FUNCTION_BLOCK PUBLIC BYTE_TO_TestSuite EXTENDS TcUnit.FB_TestSuite
VAR
END_VAR

Check_BYTE_TO_BOOL_Max();
Check_BYTE_TO_BOOL_Min();
Check_BYTE_TO_BYTE_Max();
Check_BYTE_TO_BYTE_Min();
Check_BYTE_TO_WORD_Max();
Check_BYTE_TO_WORD_Min();
Check_BYTE_TO_DWORD_Max();
Check_BYTE_TO_DWORD_Min();
Check_BYTE_TO_LWORD_Max();
Check_BYTE_TO_LWORD_Min();
Check_BYTE_TO_SINT_Max();
Check_BYTE_TO_SINT_Min();
Check_BYTE_TO_SINT_TooHigh();
Check_BYTE_TO_INT_Max();
Check_BYTE_TO_INT_Min();
Check_BYTE_TO_DINT_Max();
Check_BYTE_TO_DINT_Min();
Check_BYTE_TO_LINT_Max();
Check_BYTE_TO_LINT_Min();
Check_BYTE_TO_USINT_Max();
Check_BYTE_TO_USINT_Min();
Check_BYTE_TO_UINT_Max();
Check_BYTE_TO_UINT_Min();
Check_BYTE_TO_UDINT_Max();
Check_BYTE_TO_UDINT_Min();
Check_BYTE_TO_ULINT_Max();
Check_BYTE_TO_ULINT_Min();
Check_BYTE_TO_REAL_Max();
Check_BYTE_TO_REAL_Min();
Check_BYTE_TO_LREAL_Max();
Check_BYTE_TO_LREAL_Min();
Check_BYTE_TO_TIME_Max();
Check_BYTE_TO_TIME_Min();
Check_BYTE_TO_TOD_Max();
Check_BYTE_TO_TOD_Min();
Check_BYTE_TO_DATE_Max();
Check_BYTE_TO_DATE_Min();
Check_BYTE_TO_DT_Max();
Check_BYTE_TO_DT_Min();
Check_BYTE_TO_STRING_Max();
Check_BYTE_TO_STRING_Min();

METHOD PUBLIC Check_BYTE_TO_BOOL_Min
VAR
	value : BYTE := DatatypeLimits.BYTE_MIN_VALUE;
	actual : BOOL;
	converted : BOOL;
	equal : BOOL;
END_VAR
TEST('Check_BYTE_TO_BOOL_Min');

// @TEST-RUN
converted := TryConvert_BYTE_TO_Destination(value, actual);
equal := actual = BYTE_TO_BOOL(value);

// @TEST-ASSERT
AssertTrue(Condition := equal, Message := 'Did not convert BYTE to BOOL correctly');
AssertTrue(Condition := converted, Message := 'Did not report BYTE to BOOL conversion was successful');

TEST_FINISHED();
END_METHOD

METHOD PUBLIC Check_BYTE_TO_BOOL_Max
VAR
	value : BYTE := DatatypeLimits.BYTE_MAX_VALUE;
	actual : BOOL;
	converted : BOOL;
	equal : BOOL;
END_VAR
TEST('Check_BYTE_TO_BOOL_Max');

// @TEST-RUN
converted := TryConvert_BYTE_TO_Destination(value, actual);
equal := actual = BYTE_TO_BOOL(value);

// @TEST-ASSERT
AssertTrue(Condition := equal, Message := 'Did not convert BYTE to BOOL correctly');
AssertTrue(Condition := converted, Message := 'Did not report BYTE to BOOL conversion was successful');

TEST_FINISHED();
END_METHOD

METHOD PUBLIC Check_BYTE_TO_BYTE_Min
VAR
	value : BYTE := DatatypeLimits.BYTE_MIN_VALUE;
	actual : BYTE;
	converted : BOOL;
	equal : BOOL;
END_VAR
TEST('Check_BYTE_TO_BYTE_Min');

// @TEST-RUN
converted := TryConvert_BYTE_TO_Destination(value, actual);
equal := actual = value;

// @TEST-ASSERT
AssertTrue(Condition := equal, Message := 'Did not convert BYTE to BYTE correctly');
AssertTrue(Condition := converted, Message := 'Did not report BYTE to BYTE conversion was successful');

TEST_FINISHED();
END_METHOD

METHOD PUBLIC Check_BYTE_TO_BYTE_Max
VAR
	value : BYTE := DatatypeLimits.BYTE_MAX_VALUE;
	actual : BYTE;
	converted : BOOL;
	equal : BOOL;
END_VAR
TEST('Check_BYTE_TO_BYTE_Max');

// @TEST-RUN
converted := TryConvert_BYTE_TO_Destination(value, actual);
equal := actual = value;

// @TEST-ASSERT
AssertTrue(Condition := equal, Message := 'Did not convert BYTE to BYTE correctly');
AssertTrue(Condition := converted, Message := 'Did not report BYTE to BYTE conversion was successful');

TEST_FINISHED();
END_METHOD

METHOD PUBLIC Check_BYTE_TO_DATE_Min
VAR
	value : BYTE := DatatypeLimits.BYTE_MIN_VALUE;
	actual : DATE;
	converted : BOOL;
	equal : BOOL;
END_VAR
TEST('Check_BYTE_TO_DATE_Min');

// @TEST-RUN
converted := TryConvert_BYTE_TO_Destination(value, actual);
equal := actual = BYTE_TO_DATE(value);

// @TEST-ASSERT
AssertTrue(Condition := equal, Message := 'Did not convert BYTE to DATE correctly');
AssertTrue(Condition := converted, Message := 'Did not report BYTE to DATE conversion was successful');

TEST_FINISHED();
END_METHOD

METHOD PUBLIC Check_BYTE_TO_DATE_Max
VAR
	value : BYTE := DatatypeLimits.BYTE_MAX_VALUE;
	actual : DATE;
	converted : BOOL;
	equal : BOOL;
END_VAR
TEST('Check_BYTE_TO_DATE_Max');

// @TEST-RUN
converted := TryConvert_BYTE_TO_Destination(value, actual);
equal := actual = BYTE_TO_DATE(value);

// @TEST-ASSERT
AssertTrue(Condition := equal, Message := 'Did not convert BYTE to DATE correctly');
AssertTrue(Condition := converted, Message := 'Did not report BYTE to DATE conversion was successful');

TEST_FINISHED();
END_METHOD

METHOD PUBLIC Check_BYTE_TO_DINT_Min
VAR
	value : BYTE := DatatypeLimits.BYTE_MIN_VALUE;
	actual : DINT;
	converted : BOOL;
	equal : BOOL;
END_VAR
TEST('Check_BYTE_TO_DINT_Min');

// @TEST-RUN
converted := TryConvert_BYTE_TO_Destination(value, actual);
equal := actual = BYTE_TO_DINT(value);

// @TEST-ASSERT
AssertTrue(Condition := equal, Message := 'Did not convert BYTE to DINT correctly');
AssertTrue(Condition := converted, Message := 'Did not report BYTE to DINT conversion was successful');

TEST_FINISHED();
END_METHOD

METHOD PUBLIC Check_BYTE_TO_DINT_Max
VAR
	value : BYTE := DatatypeLimits.BYTE_MAX_VALUE;
	actual : DINT;
	converted : BOOL;
	equal : BOOL;
END_VAR
TEST('Check_BYTE_TO_DINT_Max');

// @TEST-RUN
converted := TryConvert_BYTE_TO_Destination(value, actual);
equal := actual = BYTE_TO_DINT(value);

// @TEST-ASSERT
AssertTrue(Condition := equal, Message := 'Did not convert BYTE to DINT correctly');
AssertTrue(Condition := converted, Message := 'Did not report BYTE to DINT conversion was successful');

TEST_FINISHED();
END_METHOD

METHOD PUBLIC Check_BYTE_TO_DT_Min
VAR
	value : BYTE := DatatypeLimits.BYTE_MIN_VALUE;
	actual : DT;
	converted : BOOL;
	equal : BOOL;
END_VAR
TEST('Check_BYTE_TO_DT_Min');

// @TEST-RUN
converted := TryConvert_BYTE_TO_Destination(value, actual);
equal := actual = BYTE_TO_DT(value);

// @TEST-ASSERT
AssertTrue(Condition := equal, Message := 'Did not convert BYTE to DT correctly');
AssertTrue(Condition := converted, Message := 'Did not report BYTE to DT conversion was successful');

TEST_FINISHED();
END_METHOD

METHOD PUBLIC Check_BYTE_TO_DT_Max
VAR
	value : BYTE := DatatypeLimits.BYTE_MAX_VALUE;
	actual : DT;
	converted : BOOL;
	equal : BOOL;
END_VAR
TEST('Check_BYTE_TO_DT_Max');

// @TEST-RUN
converted := TryConvert_BYTE_TO_Destination(value, actual);
equal := actual = BYTE_TO_DT(value);

// @TEST-ASSERT
AssertTrue(Condition := equal, Message := 'Did not convert BYTE to DT correctly');
AssertTrue(Condition := converted, Message := 'Did not report BYTE to DT conversion was successful');

TEST_FINISHED();
END_METHOD

METHOD PUBLIC Check_BYTE_TO_DWORD_Min
VAR
	value : BYTE := DatatypeLimits.BYTE_MIN_VALUE;
	actual : DWORD;
	converted : BOOL;
	equal : BOOL;
END_VAR
TEST('Check_BYTE_TO_DWORD_Min');

// @TEST-RUN
converted := TryConvert_BYTE_TO_Destination(value, actual);
equal := actual = BYTE_TO_DWORD(value);

// @TEST-ASSERT
AssertTrue(Condition := equal, Message := 'Did not convert BYTE to DWORD correctly');
AssertTrue(Condition := converted, Message := 'Did not report BYTE to DWORD conversion was successful');

TEST_FINISHED();
END_METHOD

METHOD PUBLIC Check_BYTE_TO_DWORD_Max
VAR
	value : BYTE := DatatypeLimits.BYTE_MAX_VALUE;
	actual : DWORD;
	converted : BOOL;
	equal : BOOL;
END_VAR
TEST('Check_BYTE_TO_DWORD_Max');

// @TEST-RUN
converted := TryConvert_BYTE_TO_Destination(value, actual);
equal := actual = BYTE_TO_DWORD(value);

// @TEST-ASSERT
AssertTrue(Condition := equal, Message := 'Did not convert BYTE to DWORD correctly');
AssertTrue(Condition := converted, Message := 'Did not report BYTE to DWORD conversion was successful');

TEST_FINISHED();
END_METHOD

METHOD PUBLIC Check_BYTE_TO_INT_Min
VAR
	value : BYTE := DatatypeLimits.BYTE_MIN_VALUE;
	actual : INT;
	converted : BOOL;
	equal : BOOL;
END_VAR
TEST('Check_BYTE_TO_INT_Min');

// @TEST-RUN
converted := TryConvert_BYTE_TO_Destination(value, actual);
equal := actual = BYTE_TO_INT(value);

// @TEST-ASSERT
AssertTrue(Condition := equal, Message := 'Did not convert BYTE to INT correctly');
AssertTrue(Condition := converted, Message := 'Did not report BYTE to INT conversion was successful');

TEST_FINISHED();
END_METHOD

METHOD PUBLIC Check_BYTE_TO_INT_Max
VAR
	value : BYTE := DatatypeLimits.BYTE_MAX_VALUE;
	actual : INT;
	converted : BOOL;
	equal : BOOL;
END_VAR
TEST('Check_BYTE_TO_INT_Max');

// @TEST-RUN
converted := TryConvert_BYTE_TO_Destination(value, actual);
equal := actual = BYTE_TO_INT(value);

// @TEST-ASSERT
AssertTrue(Condition := equal, Message := 'Did not convert BYTE to INT correctly');
AssertTrue(Condition := converted, Message := 'Did not report BYTE to INT conversion was successful');

TEST_FINISHED();
END_METHOD

METHOD PUBLIC Check_BYTE_TO_LINT_Min
VAR
	value : BYTE := DatatypeLimits.BYTE_MIN_VALUE;
	actual : LINT;
	converted : BOOL;
	equal : BOOL;
END_VAR
TEST('Check_BYTE_TO_LINT_Min');

// @TEST-RUN
converted := TryConvert_BYTE_TO_Destination(value, actual);
equal := actual = BYTE_TO_LINT(value);

// @TEST-ASSERT
AssertTrue(Condition := equal, Message := 'Did not convert BYTE to LINT correctly');
AssertTrue(Condition := converted, Message := 'Did not report BYTE to LINT conversion was successful');

TEST_FINISHED();
END_METHOD

METHOD PUBLIC Check_BYTE_TO_LINT_Max
VAR
	value : BYTE := DatatypeLimits.BYTE_MAX_VALUE;
	actual : LINT;
	converted : BOOL;
	equal : BOOL;
END_VAR
TEST('Check_BYTE_TO_LINT_Max');

// @TEST-RUN
converted := TryConvert_BYTE_TO_Destination(value, actual);
equal := actual = BYTE_TO_LINT(value);

// @TEST-ASSERT
AssertTrue(Condition := equal, Message := 'Did not convert BYTE to LINT correctly');
AssertTrue(Condition := converted, Message := 'Did not report BYTE to LINT conversion was successful');

TEST_FINISHED();
END_METHOD

METHOD PUBLIC Check_BYTE_TO_LREAL_Min
VAR
	value : BYTE := DatatypeLimits.BYTE_MIN_VALUE;
	actual : LREAL;
	converted : BOOL;
	equal : BOOL;
END_VAR
TEST('Check_BYTE_TO_LREAL_Min');

// @TEST-RUN
converted := TryConvert_BYTE_TO_Destination(value, actual);
equal := actual = BYTE_TO_LREAL(value);

// @TEST-ASSERT
AssertTrue(Condition := equal, Message := 'Did not convert BYTE to LREAL correctly');
AssertTrue(Condition := converted, Message := 'Did not report BYTE to LREAL conversion was successful');

TEST_FINISHED();
END_METHOD

METHOD PUBLIC Check_BYTE_TO_LREAL_Max
VAR
	value : BYTE := DatatypeLimits.BYTE_MAX_VALUE;
	actual : LREAL;
	converted : BOOL;
	equal : BOOL;
END_VAR
TEST('Check_BYTE_TO_LREAL_Max');

// @TEST-RUN
converted := TryConvert_BYTE_TO_Destination(value, actual);
equal := actual = BYTE_TO_LREAL(value);

// @TEST-ASSERT
AssertTrue(Condition := equal, Message := 'Did not convert BYTE to LREAL correctly');
AssertTrue(Condition := converted, Message := 'Did not report BYTE to LREAL conversion was successful');

TEST_FINISHED();
END_METHOD

METHOD PUBLIC Check_BYTE_TO_LWORD_Min
VAR
	value : BYTE := DatatypeLimits.BYTE_MIN_VALUE;
	actual : LWORD;
	converted : BOOL;
	equal : BOOL;
END_VAR
TEST('Check_BYTE_TO_LWORD_Min');

// @TEST-RUN
converted := TryConvert_BYTE_TO_Destination(value, actual);
equal := actual = BYTE_TO_LWORD(value);

// @TEST-ASSERT
AssertTrue(Condition := equal, Message := 'Did not convert BYTE to LWORD correctly');
AssertTrue(Condition := converted, Message := 'Did not report BYTE to LWORD conversion was successful');

TEST_FINISHED();
END_METHOD

METHOD PUBLIC Check_BYTE_TO_LWORD_Max
VAR
	value : BYTE := DatatypeLimits.BYTE_MAX_VALUE;
	actual : LWORD;
	converted : BOOL;
	equal : BOOL;
END_VAR
TEST('Check_BYTE_TO_LWORD_Max');

// @TEST-RUN
converted := TryConvert_BYTE_TO_Destination(value, actual);
equal := actual = BYTE_TO_LWORD(value);

// @TEST-ASSERT
AssertTrue(Condition := equal, Message := 'Did not convert BYTE to LWORD correctly');
AssertTrue(Condition := converted, Message := 'Did not report BYTE to LWORD conversion was successful');

TEST_FINISHED();
END_METHOD

METHOD PUBLIC Check_BYTE_TO_REAL_Min
VAR
	value : BYTE := DatatypeLimits.BYTE_MIN_VALUE;
	actual : REAL;
	converted : BOOL;
	equal : BOOL;
END_VAR
TEST('Check_BYTE_TO_REAL_Min');

// @TEST-RUN
converted := TryConvert_BYTE_TO_Destination(value, actual);
equal := actual = BYTE_TO_REAL(value);

// @TEST-ASSERT
AssertTrue(Condition := equal, Message := 'Did not convert BYTE to REAL correctly');
AssertTrue(Condition := converted, Message := 'Did not report BYTE to REAL conversion was successful');

TEST_FINISHED();
END_METHOD

METHOD PUBLIC Check_BYTE_TO_REAL_Max
VAR
	value : BYTE := DatatypeLimits.BYTE_MAX_VALUE;
	actual : REAL;
	converted : BOOL;
	equal : BOOL;
END_VAR
TEST('Check_BYTE_TO_REAL_Max');

// @TEST-RUN
converted := TryConvert_BYTE_TO_Destination(value, actual);
equal := actual = BYTE_TO_REAL(value);

// @TEST-ASSERT
AssertTrue(Condition := equal, Message := 'Did not convert BYTE to REAL correctly');
AssertTrue(Condition := converted, Message := 'Did not report BYTE to REAL conversion was successful');

TEST_FINISHED();
END_METHOD

METHOD PUBLIC Check_BYTE_TO_SINT_Min
VAR
	value : BYTE := DatatypeLimits.BYTE_MIN_VALUE;
	actual : SINT;
	converted : BOOL;
	equal : BOOL;
END_VAR
TEST('Check_BYTE_TO_SINT_Min');

// @TEST-RUN
converted := TryConvert_BYTE_TO_Destination(value, actual);
equal := actual = BYTE_TO_SINT(value);

// @TEST-ASSERT
AssertTrue(Condition := equal, Message := 'Did not convert BYTE to SINT correctly');
AssertTrue(Condition := converted, Message := 'Did not report BYTE to SINT conversion was successful');

TEST_FINISHED();
END_METHOD

METHOD PUBLIC Check_BYTE_TO_SINT_TooHigh
VAR
	value : BYTE := DatatypeLimits.BYTE_MAX_VALUE;
	actual : SINT;
	converted : BOOL;
END_VAR
TEST('Check_BYTE_TO_SINT_TooHigh');

// @TEST-RUN
converted := TryConvert_BYTE_TO_Destination(value, actual);

// @TEST-ASSERT
AssertFalse(Condition := converted, Message := 'Did not report BYTE to SINT conversion was prevented');

TEST_FINISHED();
END_METHOD

METHOD PUBLIC Check_BYTE_TO_SINT_Max
VAR
	value : BYTE := DatatypeLimits.MAX_VALUE_OF_BYTE_WHICH_CAN_BE_HELD_IN_A_SINT;
	actual : SINT;
	converted : BOOL;
	equal : BOOL;
END_VAR
TEST('Check_BYTE_TO_SINT_Max');

// @TEST-RUN
converted := TryConvert_BYTE_TO_Destination(value, actual);
equal := actual = BYTE_TO_SINT(value);

// @TEST-ASSERT
AssertTrue(Condition := equal, Message := 'Did not convert BYTE to SINT correctly');
AssertTrue(Condition := converted, Message := 'Did not report BYTE to SINT conversion was successful');

TEST_FINISHED();
END_METHOD

METHOD PUBLIC Check_BYTE_TO_STRING_Min
VAR
	value : BYTE := DatatypeLimits.BYTE_MIN_VALUE;
	actual : STRING;
	converted : BOOL;
	equal : BOOL;
END_VAR
TEST('Check_BYTE_TO_STRING_Min');

// @TEST-RUN
converted := TryConvert_BYTE_TO_Destination(value, actual);
equal := actual = BYTE_TO_STRING(value);

// @TEST-ASSERT
AssertTrue(Condition := equal, Message := 'Did not convert BYTE to STRING correctly');
AssertTrue(Condition := converted, Message := 'Did not report BYTE to STRING conversion was successful');

TEST_FINISHED();
END_METHOD

METHOD PUBLIC Check_BYTE_TO_STRING_Max
VAR
	value : BYTE := DatatypeLimits.BYTE_MAX_VALUE;
	actual : STRING;
	converted : BOOL;
	equal : BOOL;
END_VAR
TEST('Check_BYTE_TO_STRING_Max');

// @TEST-RUN
converted := TryConvert_BYTE_TO_Destination(value, actual);
equal := actual = BYTE_TO_STRING(value);

// @TEST-ASSERT
AssertTrue(Condition := equal, Message := 'Did not convert BYTE to STRING correctly');
AssertTrue(Condition := converted, Message := 'Did not report BYTE to STRING conversion was successful');

TEST_FINISHED();
END_METHOD

METHOD PUBLIC Check_BYTE_TO_TIME_Min
VAR
	value : BYTE := DatatypeLimits.BYTE_MIN_VALUE;
	actual : TIME;
	converted : BOOL;
	equal : BOOL;
END_VAR
TEST('Check_BYTE_TO_TIME_Min');

// @TEST-RUN
converted := TryConvert_BYTE_TO_Destination(value, actual);
equal := actual = BYTE_TO_TIME(value);

// @TEST-ASSERT
AssertTrue(Condition := equal, Message := 'Did not convert BYTE to TIME correctly');
AssertTrue(Condition := converted, Message := 'Did not report BYTE to TIME conversion was successful');

TEST_FINISHED();
END_METHOD

METHOD PUBLIC Check_BYTE_TO_TIME_Max
VAR
	value : BYTE := DatatypeLimits.BYTE_MAX_VALUE;
	actual : TIME;
	converted : BOOL;
	equal : BOOL;
END_VAR
TEST('Check_BYTE_TO_TIME_Max');

// @TEST-RUN
converted := TryConvert_BYTE_TO_Destination(value, actual);
equal := actual = BYTE_TO_TIME(value);

// @TEST-ASSERT
AssertTrue(Condition := equal, Message := 'Did not convert BYTE to TIME correctly');
AssertTrue(Condition := converted, Message := 'Did not report BYTE to TIME conversion was successful');

TEST_FINISHED();
END_METHOD

METHOD PUBLIC Check_BYTE_TO_TOD_Min
VAR
	value : BYTE := DatatypeLimits.BYTE_MIN_VALUE;
	actual : TOD;
	converted : BOOL;
	equal : BOOL;
END_VAR
TEST('Check_BYTE_TO_TOD_Min');

// @TEST-RUN
converted := TryConvert_BYTE_TO_Destination(value, actual);
equal := actual = BYTE_TO_TOD(value);

// @TEST-ASSERT
AssertTrue(Condition := equal, Message := 'Did not convert BYTE to TOD correctly');
AssertTrue(Condition := converted, Message := 'Did not report BYTE to TOD conversion was successful');

TEST_FINISHED();
END_METHOD

METHOD PUBLIC Check_BYTE_TO_TOD_Max
VAR
	value : BYTE := DatatypeLimits.BYTE_MAX_VALUE;
	actual : TOD;
	converted : BOOL;
	equal : BOOL;
END_VAR
TEST('Check_BYTE_TO_TOD_Max');

// @TEST-RUN
converted := TryConvert_BYTE_TO_Destination(value, actual);
equal := actual = BYTE_TO_TOD(value);

// @TEST-ASSERT
AssertTrue(Condition := equal, Message := 'Did not convert BYTE to TOD correctly');
AssertTrue(Condition := converted, Message := 'Did not report BYTE to TOD conversion was successful');

TEST_FINISHED();
END_METHOD

METHOD PUBLIC Check_BYTE_TO_UDINT_Min
VAR
	value : BYTE := DatatypeLimits.BYTE_MIN_VALUE;
	actual : UDINT;
	converted : BOOL;
	equal : BOOL;
END_VAR
TEST('Check_BYTE_TO_UDINT_Min');

// @TEST-RUN
converted := TryConvert_BYTE_TO_Destination(value, actual);
equal := actual = BYTE_TO_UDINT(value);

// @TEST-ASSERT
AssertTrue(Condition := equal, Message := 'Did not convert BYTE to UDINT correctly');
AssertTrue(Condition := converted, Message := 'Did not report BYTE to UDINT conversion was successful');

TEST_FINISHED();
END_METHOD

METHOD PUBLIC Check_BYTE_TO_UDINT_Max
VAR
	value : BYTE := DatatypeLimits.BYTE_MAX_VALUE;
	actual : UDINT;
	converted : BOOL;
	equal : BOOL;
END_VAR
TEST('Check_BYTE_TO_UDINT_Max');

// @TEST-RUN
converted := TryConvert_BYTE_TO_Destination(value, actual);
equal := actual = BYTE_TO_UDINT(value);

// @TEST-ASSERT
AssertTrue(Condition := equal, Message := 'Did not convert BYTE to UDINT correctly');
AssertTrue(Condition := converted, Message := 'Did not report BYTE to UDINT conversion was successful');

TEST_FINISHED();
END_METHOD

METHOD PUBLIC Check_BYTE_TO_UINT_Min
VAR
	value : BYTE := DatatypeLimits.BYTE_MIN_VALUE;
	actual : UINT;
	converted : BOOL;
	equal : BOOL;
END_VAR
TEST('Check_BYTE_TO_UINT_Min');

// @TEST-RUN
converted := TryConvert_BYTE_TO_Destination(value, actual);
equal := actual = BYTE_TO_UINT(value);

// @TEST-ASSERT
AssertTrue(Condition := equal, Message := 'Did not convert BYTE to UINT correctly');
AssertTrue(Condition := converted, Message := 'Did not report BYTE to UINT conversion was successful');

TEST_FINISHED();
END_METHOD

METHOD PUBLIC Check_BYTE_TO_UINT_Max
VAR
	value : BYTE := DatatypeLimits.BYTE_MAX_VALUE;
	actual : UINT;
	converted : BOOL;
	equal : BOOL;
END_VAR
TEST('Check_BYTE_TO_UINT_Max');

// @TEST-RUN
converted := TryConvert_BYTE_TO_Destination(value, actual);
equal := actual = BYTE_TO_UINT(value);

// @TEST-ASSERT
AssertTrue(Condition := equal, Message := 'Did not convert BYTE to UINT correctly');
AssertTrue(Condition := converted, Message := 'Did not report BYTE to UINT conversion was successful');

TEST_FINISHED();
END_METHOD

METHOD PUBLIC Check_BYTE_TO_ULINT_Min
VAR
	value : BYTE := DatatypeLimits.BYTE_MIN_VALUE;
	actual : ULINT;
	converted : BOOL;
	equal : BOOL;
END_VAR
TEST('Check_BYTE_TO_ULINT_Min');

// @TEST-RUN
converted := TryConvert_BYTE_TO_Destination(value, actual);
equal := actual = BYTE_TO_ULINT(value);

// @TEST-ASSERT
AssertTrue(Condition := equal, Message := 'Did not convert BYTE to ULINT correctly');
AssertTrue(Condition := converted, Message := 'Did not report BYTE to ULINT conversion was successful');

TEST_FINISHED();
END_METHOD

METHOD PUBLIC Check_BYTE_TO_ULINT_Max
VAR
	value : BYTE := DatatypeLimits.BYTE_MAX_VALUE;
	actual : ULINT;
	converted : BOOL;
	equal : BOOL;
END_VAR
TEST('Check_BYTE_TO_ULINT_Max');

// @TEST-RUN
converted := TryConvert_BYTE_TO_Destination(value, actual);
equal := actual = BYTE_TO_ULINT(value);

// @TEST-ASSERT
AssertTrue(Condition := equal, Message := 'Did not convert BYTE to ULINT correctly');
AssertTrue(Condition := converted, Message := 'Did not report BYTE to ULINT conversion was successful');

TEST_FINISHED();
END_METHOD

METHOD PUBLIC Check_BYTE_TO_USINT_Min
VAR
	value : BYTE := DatatypeLimits.BYTE_MIN_VALUE;
	actual : USINT;
	converted : BOOL;
	equal : BOOL;
END_VAR
TEST('Check_BYTE_TO_USINT_Min');

// @TEST-RUN
converted := TryConvert_BYTE_TO_Destination(value, actual);
equal := actual = BYTE_TO_USINT(value);

// @TEST-ASSERT
AssertTrue(Condition := equal, Message := 'Did not convert BYTE to USINT correctly');
AssertTrue(Condition := converted, Message := 'Did not report BYTE to USINT conversion was successful');

TEST_FINISHED();
END_METHOD

METHOD PUBLIC Check_BYTE_TO_USINT_Max
VAR
	value : BYTE := DatatypeLimits.BYTE_MAX_VALUE;
	actual : USINT;
	converted : BOOL;
	equal : BOOL;
END_VAR
TEST('Check_BYTE_TO_USINT_Max');

// @TEST-RUN
converted := TryConvert_BYTE_TO_Destination(value, actual);
equal := actual = BYTE_TO_USINT(value);

// @TEST-ASSERT
AssertTrue(Condition := equal, Message := 'Did not convert BYTE to USINT correctly');
AssertTrue(Condition := converted, Message := 'Did not report BYTE to USINT conversion was successful');

TEST_FINISHED();
END_METHOD

METHOD PUBLIC Check_BYTE_TO_WORD_Min
VAR
	value : BYTE := DatatypeLimits.BYTE_MIN_VALUE;
	actual : WORD;
	converted : BOOL;
	equal : BOOL;
END_VAR
TEST('Check_BYTE_TO_WORD_Min');

// @TEST-RUN
converted := TryConvert_BYTE_TO_Destination(value, actual);
equal := actual = BYTE_TO_WORD(value);

// @TEST-ASSERT
AssertTrue(Condition := equal, Message := 'Did not convert BYTE to WORD correctly');
AssertTrue(Condition := converted, Message := 'Did not report BYTE to WORD conversion was successful');

TEST_FINISHED();
END_METHOD

METHOD PUBLIC Check_BYTE_TO_WORD_Max
VAR
	value : BYTE := DatatypeLimits.BYTE_MAX_VALUE;
	actual : WORD;
	converted : BOOL;
	equal : BOOL;
END_VAR
TEST('Check_BYTE_TO_WORD_Max');

// @TEST-RUN
converted := TryConvert_BYTE_TO_Destination(value, actual);
equal := actual = BYTE_TO_WORD(value);

// @TEST-ASSERT
AssertTrue(Condition := equal, Message := 'Did not convert BYTE to WORD correctly');
AssertTrue(Condition := converted, Message := 'Did not report BYTE to WORD conversion was successful');

TEST_FINISHED();
END_METHOD

END_FUNCTION_BLOCK

(* stored: Version 1.1.0.1, ProductVersion 3.1.4024.12
   POU BYTE_TO_TestSuite: Id {c38927c0-9683-4451-b3bb-c40c98c84496}, SpecialFunc None
   Method Check_BYTE_TO_BOOL_Min: Id {ac87d2f6-db36-43f6-a7e2-3782b29cdbe9}
   Method Check_BYTE_TO_BOOL_Max: Id {0b2bb98c-65c5-4fde-89f8-a39c52c26978}
   Method Check_BYTE_TO_BYTE_Min: Id {f6660d92-b1e3-4bd7-859e-bdf26e62f002}
   Method Check_BYTE_TO_BYTE_Max: Id {214aa7e3-4abb-4d75-9c99-83868509447e}
   Method Check_BYTE_TO_DATE_Min: Id {320bf2d8-ca67-46f1-ba33-720bd20321f8}
   Method Check_BYTE_TO_DATE_Max: Id {3cf17eab-74ac-46e2-a95f-2c07971ee139}
   Method Check_BYTE_TO_DINT_Min: Id {e508eea2-52a0-40ff-9ef8-14ae11ecc757}
   Method Check_BYTE_TO_DINT_Max: Id {bfe0cd31-916e-4fd6-947b-d5c0748704be}
   Method Check_BYTE_TO_DT_Min: Id {81196007-2d5a-43ab-b4fc-58fdaa84fc8d}
   Method Check_BYTE_TO_DT_Max: Id {a684ce64-9c59-42db-a531-1c0930e01ec0}
   Method Check_BYTE_TO_DWORD_Min: Id {ceda0525-c609-4a2b-91c9-dfd57021404f}
   Method Check_BYTE_TO_DWORD_Max: Id {394ec300-8e92-4750-a92d-f5a449afe173}
   Method Check_BYTE_TO_INT_Min: Id {8080f2f9-d096-4f16-88b2-2f50c8ec5a75}
   Method Check_BYTE_TO_INT_Max: Id {c6146aec-040c-41b1-99b7-e81a82ec74bb}
   Method Check_BYTE_TO_LINT_Min: Id {d2a15a3c-8591-41c6-8f8a-712b75da87ca}
   Method Check_BYTE_TO_LINT_Max: Id {715385c8-ee4f-4666-b813-06813d334745}
   Method Check_BYTE_TO_LREAL_Min: Id {4a6da61f-ab07-4d60-b4f7-770e1b95f180}
   Method Check_BYTE_TO_LREAL_Max: Id {13263a4d-bed1-4e61-a453-3e2a16e91009}
   Method Check_BYTE_TO_LWORD_Min: Id {5e4906f1-9173-415e-8d6f-9de78ecf07e0}
   Method Check_BYTE_TO_LWORD_Max: Id {b8d892bc-5a1a-4f94-a867-37a708170076}
   Method Check_BYTE_TO_REAL_Min: Id {66d88623-6280-4b85-81db-00980d11a0d7}
   Method Check_BYTE_TO_REAL_Max: Id {833c93a5-b68d-4efc-8c07-64ad0e2f0534}
   Method Check_BYTE_TO_SINT_Min: Id {fc3c69e3-2268-4748-a95b-d54e6dac5486}
   Method Check_BYTE_TO_SINT_TooHigh: Id {4f82368a-ed93-4eda-a2df-8a1a25520103}
   Method Check_BYTE_TO_SINT_Max: Id {7662b3d2-9f21-4887-9d3f-1fba962bb068}
   Method Check_BYTE_TO_STRING_Min: Id {3b139635-c449-4125-bcae-96bc5cb96dfa}
   Method Check_BYTE_TO_STRING_Max: Id {1dfa0191-b3fa-40c4-b43e-69cf43fff885}
   Method Check_BYTE_TO_TIME_Min: Id {cc87951f-0127-41f4-9ae6-8f9b79fe08d3}
   Method Check_BYTE_TO_TIME_Max: Id {48ed6b00-2296-4db2-b5ae-ff0138cc5110}
   Method Check_BYTE_TO_TOD_Min: Id {867e7ef4-4226-4fdd-bd7b-8f696c0a4ba9}
   Method Check_BYTE_TO_TOD_Max: Id {fefb83ce-cd15-4fba-804b-3fb377456bc0}
   Method Check_BYTE_TO_UDINT_Min: Id {105ca9eb-1da0-4753-9a84-b70159b2c3d5}
   Method Check_BYTE_TO_UDINT_Max: Id {5bfa05f3-8c34-4808-b049-9a95bf4cb139}
   Method Check_BYTE_TO_UINT_Min: Id {abec39c6-c70d-4eb7-a674-0c7ee202b0b4}
   Method Check_BYTE_TO_UINT_Max: Id {9b863ea2-c33a-4fd3-a6fc-46f1a04d9c6a}
   Method Check_BYTE_TO_ULINT_Min: Id {4459ea7e-e863-4bfe-a213-57bb397357e9}
   Method Check_BYTE_TO_ULINT_Max: Id {4d269956-1a5a-4223-bd85-678fc11d7cca}
   Method Check_BYTE_TO_USINT_Min: Id {466c0147-49db-4795-9fd6-3496b523087c}
   Method Check_BYTE_TO_USINT_Max: Id {c56cfcd3-4ee2-4a1a-9412-695ab5be1610}
   Method Check_BYTE_TO_WORD_Min: Id {9d24b7a5-2d36-4d60-8627-3e676ad233bc}
   Method Check_BYTE_TO_WORD_Max: Id {82b2f5e8-925d-423b-9dfb-e5c06b87b59e} *)
